{attribute 'GeneratedUsingTerminal: ELM9410-0000-0016'}
{attribute addProperty BoxType "ELM9410-0000-0016"}
{attribute addProperty Id "DiagBOOL1ErrorBOOL1Input_cycle_CounterBYTE1TxPDO_StateBOOL1"}
{attribute addProperty CRC "101989023"}
{attribute addProperty Size "4"}
TYPE Status_06143A9F :
STRUCT
	{attribute addProperty Name "Diag"}
	Diag : BOOL;
	{attribute addProperty Name "Error"}
	Error : BOOL;
	{attribute addProperty Name "Input_cycle_Counter"}
	Input_cycle_Counter : BYTE;
	{attribute addProperty Name "TxPDO_State"}
	TxPDO_State : BOOL;
END_STRUCT
END_TYPE

(* stored: Version 1.2.0.0, ProductVersion 3.1.4024.11
   DUT Status_06143A9F: Id {6b56bd03-fb24-4101-ac41-b575f0453ddf} *)
